// TIA Portal V18 export
VAR_GLOBAL   // PLC tag table "PLCIO_DQ"
   oHMIControlOn AT %Q100.0 : Bool;   // HMI_上电按钮 / HMI_Power on button
   oHMIMachineStart AT %Q100.1 : Bool;   // HMI_设备启动按钮 / HMI_Device start button
   oHMIMachineStop AT %Q100.2 : Bool;   // HMI_设备停止按钮 / HMI_Device Stop Button
   oHMIResetButton AT %Q100.3 : Bool;   // HMI_复位按钮 / HMI_reset button
   oHMISafetyGateUnlock AT %Q100.4 : Bool;   // HMI_安全门解锁按钮 / HMI_safety door unlock button
   "RESERVE_Q100.5" AT %Q100.5 : Bool;   // 备用_Q100.5 / Spare_Q100.5
   "RESERVE_Q100.6" AT %Q100.6 : Bool;   // 备用_Q100.6 / Standby_Q100.6
   "RESERVE_Q100.7" AT %Q100.7 : Bool;   // 备用_Q100.7 / Standby_Q100.7
   "oTowerLight-Green" AT %Q101.0 : Bool;   // 稳光-绿 / Steady light-green
   "oTowerLight-Red" AT %Q101.1 : Bool;   // 稳光-红 / Steady Light-Red
   "oTowerLight-yellow" AT %Q101.2 : Bool;   // 稳光-黄 / Stable light-yellow
   "oTowerLight-Blue" AT %Q101.3 : Bool;   // 稳光-蓝 / Steady Light-Blue
   "oTowerLight-Buzzer" AT %Q101.4 : Bool;   // 蜂鸣 / buzz
   oLED_lamp_1 AT %Q101.5 : Bool;   // 日光灯_1 / Fluorescent lamp_1
   oLED_lamp_2 AT %Q101.6 : Bool;   // 日光灯_2 / Fluorescent lamp_2
   oSafetyPLC AT %Q101.7 : Bool;   // 安全PLC / Safety PLC
   oSafetyDoorLocked_1 AT %Q102.0 : Bool;   // 安全门锁定_1 / Security door lock_1
   oSafetyDoorLocked_2 AT %Q102.1 : Bool;   // 安全门锁定_2 / Security door lock_2
   oSafetyDoorLocked_3 AT %Q102.2 : Bool;   // 安全门锁定_3 / Security door lock_3
   oSafetyDoorLocked_4 AT %Q102.3 : Bool;   // 安全门锁定_4 / Security door lock_4
   oSafetyDoorLocked_5 AT %Q102.4 : Bool;   // 安全门锁定_5 / Security door lock_5
   oSafetyDoorLocked_6 AT %Q102.5 : Bool;   // 安全门锁定_6 / Security door lock_6
   oSafetyDoorLocked_7 AT %Q102.6 : Bool;   // 安全门锁定_7 / Security door lock_7
   oSafetyDoorLocked_8 AT %Q102.7 : Bool;   // 安全门锁定_8 / Security door lock_8
   oSafetyDoorLocked AT %Q103.0 : Bool;   // 连锁安全门锁定 / interlock security door lock
   "oE-NG-01SafetyGate" AT %Q103.1 : Bool;   // E-NG料盒-01安全门锁 / E-NG material box-01 safety door lock
   oMaterielDoorLocked_H2 AT %Q103.4 : Bool;   // 物料门锁定_2 / Material door lock_2
   oMaterielDoorLocked_J1 AT %Q103.5 : Bool;   // 物料门锁定_3 / Material door lock_3
   "oE-NG-02SafetyGate" AT %Q103.2 : Bool;   // E-NG料盒-02安全门锁 / E-NG material box-02 safety door lock
   oMaterielDoorLocked_H1 AT %Q103.3 : Bool;   // 物料门锁定_1 / Material door lock_1
   oMaterielDoorLocked_J2 AT %Q103.6 : Bool;   // 物料门锁定_4 / Material door lock_4
   oMaterielDoorLocked_K1 AT %Q103.7 : Bool;   // 物料门锁定_5 / Material door lock_5
   oNG_Button1 AT %Q104.0 : Bool;   // NG下料按钮1 / NG blanking button 1
   oNG_Button2 AT %Q104.1 : Bool;   // NG下料按钮2 / NG blanking button 2
   oShaft_Button AT %Q104.2 : Bool;   // shaft 上料按钮 / shaft loading button
   oShaft_EmptyButton AT %Q104.3 : Bool;   // shaft 取空料盘按钮 / shaft empty tray button
   oMagnet_Button AT %Q104.4 : Bool;   // Magnet上料按钮 / Magnet loading button
   oMagnet_EmptyButton AT %Q104.5 : Bool;   // Magnet取空料盘按钮 / Magnet empty tray button
   oMagnet_UnlockButton AT %Q104.6 : Bool;   // Magne门解锁按钮 / Magne door unlock button
   "RESERVE_Q104.7" AT %Q104.7 : Bool;   // 备用_Q104.7 / Standby_Q104.7
   oUnloading_EmptyButton AT %Q105.4 : Bool;   // Unloading取空料盘按钮 / Unloading empty tray button
   oUnloading_UnlockButton AT %Q105.5 : Bool;   // Unloading门解锁按钮 / Unloading door unlock button
   oMaterielDoorLocked_K2 AT %Q105.6 : Bool;   // 物料门锁定_6 / Material door lock_6
   oMaterielDoorLocked_L1 AT %Q105.7 : Bool;   // 物料门锁定_7 / Material door lock_7
   oReserved_Button AT %Q105.0 : Bool;   // Reserved上料按钮 / Reserved feeding button
   oReserved_EmptyButton AT %Q105.1 : Bool;   // Reserved取空料盘按钮 / Reserved empty tray button
   oReserved_UnlockButton AT %Q105.2 : Bool;   // Reserved门解锁按钮 / Reserved door unlock button
   oUnloading_Button AT %Q105.3 : Bool;   // Unloading按钮 / Unloading button
   "oC-GluingPro_X" AT %Q106.0 : Bool;   // C-涂胶模组点胶阀_a / C-gluing system programX
   "oC-GluingPro_Y" AT %Q106.1 : Bool;   // C-涂胶模组点胶阀_b / C-gluing system program Y
   "oC-GluingReset" AT %Q106.2 : Bool;   // C-涂胶模组点胶阀_c / C-Gluing system reset
   "oC-GluingPro_Z" AT %Q106.3 : Bool;   // 备用_Q106.3 / C-Glue coating system program Z
   "oH-shaftLifting_SpeedChange" AT %Q106.4 : Bool;   // H-shaft 顶升位驱动电机_速度切换 / H-shaft lifting position drive motor_speed switching
   "oH-shaftLifting_Start" AT %Q106.5 : Bool;   // H-shaft 顶升位驱动电机_启动进料 / H-shaft lifting position drive motor_start feeding
   "oJ-magnetLifting_SpeedChange" AT %Q106.6 : Bool;   // J-magnet顶升驱动电机_速度切换 / J-magnet jacking drive motor_speed switching
   "oJ-magnetLifting_Start" AT %Q106.7 : Bool;   // J-magnet顶升驱动电机_启动进料 / J-magnet jacking drive motor_start feeding
   "oK-Lifting3_SpeedChange" AT %Q107.0 : Bool;   // K-预留顶升位3驱动电机_速度切换 / K-reserved jacking position 3 drive motor_speed switching
   "oK-Lifting3_Start" AT %Q107.1 : Bool;   // K-预留顶升位3驱动电机_启动进料 / K-reserved jacking position 3 drive motor_start feeding
   "oL-Unloading_CCW" AT %Q107.2 : Bool;   // L-下料线体移栽电机_出料 / L-Blanking wire body transplanting motor_discharging
   "oL-Unloading_CW" AT %Q107.3 : Bool;   // L-下料线体移栽电机_进料 / L-Blanking wire body transplanting motor_Feeding
   "oH-shaftLifting_CCWStart" AT %Q107.4 : Bool;   // H-shaft 顶升位驱动电机_启动反转出料 / H-shaft lifting position drive motor_start reverse discharging
   "oJ-magnetLifting_CCWStart" AT %Q107.5 : Bool;   // J-magnet顶升驱动电机_启动反转出料 / J-magnet jacking drive motor_start reverse discharging
   "oK-Lifting3_CCWStart" AT %Q107.6 : Bool;   // K-预留顶升位3驱动电机_启动反转出料 / K-reserved jacking position 3 drive motor_start reverse discharging
   "RESERVE_Q107.7" AT %Q107.7 : Bool;   // 备用_Q107.7 / Standby_Q107.7
   "oH-shaftLoading_CCW" AT %Q108.0 : Bool;   // H-shaft上料线体驱动电机_反转 / H-shaft feeding line body drive motor_reverse
   "oH-shaftLoading_CW" AT %Q108.1 : Bool;   // H-shaft上料线体驱动电机_正转 / H-shaft feeding line body drive motor_forward rotation
   "oH-shaftTake_CW" AT %Q108.2 : Bool;   // H-shaft取空盘驱动电机_正转 / H-shaft empty plate drive motor_forward rotation
   "oH-shaftTake_CCW" AT %Q108.3 : Bool;   // H-shaft取空盘驱动电机_反转 / H-shaft empty plate drive motor_reverse
   "RESERVE_Q108.4" AT %Q108.4 : Bool;   // 备用_Q108.4 / Standby_Q108.4
   "RESERVE_Q108.5" AT %Q108.5 : Bool;   // 备用_Q108.5 / Standby_Q108.5
   "RESERVE_Q108.6" AT %Q108.6 : Bool;   // 备用_Q108.6 / Standby_Q108.6
   "RESERVE_Q108.7" AT %Q108.7 : Bool;   // 备用_Q108.7 / Standby_Q108.7
   "RESERVE_Q109.0" AT %Q109.0 : Bool;
   "RESERVE_Q109.1" AT %Q109.1 : Bool;
   "RESERVE_Q109.2" AT %Q109.2 : Bool;
   "RESERVE_Q109.3" AT %Q109.3 : Bool;
   "RESERVE_Q109.4" AT %Q109.4 : Bool;
   "RESERVE_Q109.5" AT %Q109.5 : Bool;
   "RESERVE_Q109.6" AT %Q109.6 : Bool;
   "RESERVE_Q109.7" AT %Q109.7 : Bool;
   "J-magnet Loading _CCW" AT %Q110.0 : Bool;   // J-magnet上料线体驱动电机_反转 / J-magnet feeding line body drive motor_reverse
   "J-magnet Loading _CW" AT %Q110.1 : Bool;   // J-magnet上料线体驱动电机_正转 / J-magnet feeding line body drive motor_forward rotation
   "J-magnet Take _CW" AT %Q110.2 : Bool;   // J-magnet取空盘驱动电机_正转 / J-magnet empty disk drive motor_forward rotation
   "J-magnet Take _CCW" AT %Q110.3 : Bool;   // J-magnet取空盘驱动电机_反转 / J-magnet empty disk drive motor_reverse
   "RESERVE_Q110.4" AT %Q110.4 : Bool;   // 备用_Q110.4 / Standby_Q110.4
   "RESERVE_Q110.5" AT %Q110.5 : Bool;   // 备用_Q110.5 / Standby_Q110.5
   "RESERVE_Q110.6" AT %Q110.6 : Bool;   // 备用_Q110.6 / Standby_Q110.6
   "RESERVE_Q110.7" AT %Q110.7 : Bool;   // 备用_Q110.7 / Standby_Q110.7
   "RESERVE_Q111.0" AT %Q111.0 : Bool;
   "RESERVE_Q111.1" AT %Q111.1 : Bool;
   "RESERVE_Q111.2" AT %Q111.2 : Bool;
   "RESERVE_Q111.3" AT %Q111.3 : Bool;
   "RESERVE_Q111.4" AT %Q111.4 : Bool;
   "RESERVE_Q111.5" AT %Q111.5 : Bool;
   "RESERVE_Q111.6" AT %Q111.6 : Bool;
   "RESERVE_Q111.7" AT %Q111.7 : Bool;
   "L-Unloading _LineMotor_CCW" AT %Q112.0 : Bool;   // K-预留上料线体驱动电机_反转 / L-Blanking line drive motor_reverse
   "L-Unloading _LineMotor_CW" AT %Q112.1 : Bool;   // K-预留上料线体驱动电机_正转 / L-Blanking wire body drive motor_True story
   "K-Take _CW" AT %Q112.2 : Bool;   // K-预留取空盘驱动电机_正转 / K-reserved empty disk drive motor_forward rotation
   "K-Take _CCW" AT %Q112.3 : Bool;   // K-预留取空盘驱动电机_反转 / K-reserved empty disk drive motor_reverse
   "RESERVE_Q112.4" AT %Q112.4 : Bool;   // 备用_Q112.4 / Standby_Q112.4
   "RESERVE_Q112.5" AT %Q112.5 : Bool;   // 备用_Q112.5 / Standby_Q112.5
   "RESERVE_Q112.6" AT %Q112.6 : Bool;   // 备用_Q112.6 / Standby_Q112.6
   "RESERVE_Q112.7" AT %Q112.7 : Bool;   // 备用_Q112.7 / Standby_Q112.7
   "RESERVE_Q113.0" AT %Q113.0 : Bool;
   "RESERVE_Q113.1" AT %Q113.1 : Bool;
   "RESERVE_Q113.2" AT %Q113.2 : Bool;
   "RESERVE_Q113.3" AT %Q113.3 : Bool;
   "RESERVE_Q113.4" AT %Q113.4 : Bool;
   "RESERVE_Q113.5" AT %Q113.5 : Bool;
   "RESERVE_Q113.6" AT %Q113.6 : Bool;
   "RESERVE_Q113.7" AT %Q113.7 : Bool;
   "K-Loading _CCW" AT %Q114.0 : Bool;   // L-下料线体驱动电机_反转 / K-reserved feeding line body drive motor_reverse
   "K-Loading _CW" AT %Q114.1 : Bool;   // L-下料线体驱动电机_正传 / K-reserved feeding line body drive motor_forward rotation
   "RESERVE_Q114.2" AT %Q114.2 : Bool;   // 备用_Q114.2 / Standby_Q114.2
   "RESERVE_Q114.3" AT %Q114.3 : Bool;   // 备用_Q114.3 / Standby_Q114.3
   "RESERVE_Q114.4" AT %Q114.4 : Bool;   // 备用_Q114.4 / Standby_Q114.4
   "RESERVE_Q114.5" AT %Q114.5 : Bool;   // 备用_Q114.5 / Standby_Q114.5
   "RESERVE_Q114.6" AT %Q114.6 : Bool;   // 备用_Q114.6 / Standby_Q114.6
   "RESERVE_Q114.7" AT %Q114.7 : Bool;   // 备用_Q114.7 / Standby_Q114.7
   "RESERVE_Q115.0" AT %Q115.0 : Bool;
   "RESERVE_Q115.1" AT %Q115.1 : Bool;
   "RESERVE_Q115.2" AT %Q115.2 : Bool;
   "RESERVE_Q115.3" AT %Q115.3 : Bool;
   "RESERVE_Q115.4" AT %Q115.4 : Bool;
   "RESERVE_Q115.5" AT %Q115.5 : Bool;
   "RESERVE_Q115.6" AT %Q115.6 : Bool;
   "RESERVE_Q115.7" AT %Q115.7 : Bool;
END_VAR
